// TwinCAT 3 PLC project PRG_B_IO
// Title: B_IO
// Company: RafalOS
// Author: Rafał Osajda
// ProjectVersion: 0.0.0.7
// ProgramVersion: 3.1.4024.0
// libraries:
//   B_Base, * (RafalOS)
//   Tc2_Standard, * (Beckhoff Automation GmbH)
//   Tc2_System, * (Beckhoff Automation GmbH)
//   Tc3_Module, * (Beckhoff Automation GmbH)
// project tree:
//   / PlcTask.TcTTO (not stored)
//   POUs Compilation/ PRG_Compilation.TcPOU (not stored)
//   POUs/Electrovalve/ E_IOElectrovalveAction.TcDUT (not stored), E_IOElectrovalveType.TcDUT (not stored), FB_IOElectrovalve.TcPOU, FB_IOElectrovalve_3on2_NC.TcPOU (not stored), FB_IOElectrovalve_3on2_NO.TcPOU (not stored), FB_IOElectrovalve_5on2_1Coil.TcPOU, FB_IOElectrovalve_5on2_2Coil.TcPOU (not stored), FB_IOElectrovalve_5on3_2Coil_Vented.TcPOU (not stored), FB_IOElectrovalve_5on3_2Coil_Infected.TcPOU (not stored), ITF_IOElectrovalve.TcIO, ITF_IOElectrovalve_HMI_Init.TcIO (not stored), ITF_IOElectrovalve_HMI_Connector.TcIO
//   POUs/Sensor/ E_IOSensorType.TcDUT, FB_IOSensor.TcPOU (not stored), FB_IOSensor_NC.TcPOU, FB_IOSensor_NO.TcPOU, FB_IOSensor_NO_2InRow.TcPOU, ITF_IOSensor.TcIO (not stored), ITF_IOSensor_HMI_Init.TcIO (not stored), ITF_IOSensor_HMI_Connector.TcIO (not stored)
//   POUs/LampkaRozszerzona/ FB_IOLampBlinking.TcPOU, ITF_IOLampBlinking.TcIO
//   POUs/Lampka/ FB_IOLamp.TcPOU (not stored), ITF_IOLamp.TcIO
//   POUs/Przyciski/ FB_IOButton.TcPOU (not stored), FB_IOButton_NC.TcPOU (not stored), FB_IOButton_NO.TcPOU (not stored), ITF_IOButton.TcIO

// ---- POUs/Sensor/E_IOSensorType.TcDUT
{attribute 'qualified_only'}
{attribute 'strict'}
TYPE E_IOSensorType :
(
	NO 		:= 0,
	NC		:= 1,
	NOx2	:= 2
);
END_TYPE

// ---- POUs/Electrovalve/ITF_IOElectrovalve.TcIO
(*
	RJM Maszyny sp. z o.o.
	autor 	: Rafał Osajda
	data	: 21.02.2024
	TC		: 3.1 4024.54
	wersja	: 0.0.1.0	: pełna obsługa

	Obsługa elektrozaworu do sterowania siłownikiem pneumatycznym
*)
INTERFACE ITF_IOElectrovalve EXTENDS ITF_BaseComponent

(*
	RJM Maszyny sp. z o.o.
	autor 	: Rafał Osajda
	data	: 21.02.2024
	TC		: 3.1 4024.54
	wersja	: 0.0.1.0	: pełna obsługa

	Ustawienie odpowiednich wyjść
*)
METHOD Contol : BOOL
VAR_INPUT
	eAction									: E_IOElectrovalveAction;
END_VAR
END_METHOD

END_INTERFACE

// ---- POUs/Electrovalve/ITF_IOElectrovalve_HMI_Connector.TcIO
INTERFACE ITF_IOElectrovalve_HMI_Connector EXTENDS ITF_BaseComponent_HMI_Connector

METHOD PUBLIC GetElectrovalveType : E_IOElectrovalveType
VAR_INPUT
END_VAR
END_METHOD

METHOD PUBLIC GetElectrovalveTypeToString : STRING
END_METHOD

METHOD IsActiveCoilA : BOOL
VAR_INPUT
END_VAR
END_METHOD

METHOD IsActiveCoilB : BOOL
VAR_INPUT
END_VAR
END_METHOD

END_INTERFACE

// ---- POUs/LampkaRozszerzona/ITF_IOLampBlinking.TcIO
INTERFACE ITF_IOLampBlinking EXTENDS ITF_IOLamp

(*			
	EVERDE sp. z o.o.
	Rafał Osajda		31.01.2025		TC 4026.13		wer. 0.0.0.1
	Sterowanie działem ipulsatora 
*)
METHOD PUBLIC SetBlink
VAR_INPUT
	bIN				: bool;
END_VAR
END_METHOD

(*			
	EVERDE sp. z o.o.
	Rafał Osajda		31.01.2025		TC 4026.13		wer. 0.0.0.1
	Ustawia czas zgaszonej lampki
*)
METHOD PUBLIC SetTimeOff
VAR_INPUT
	rIN					: REAL;
END_VAR
END_METHOD

(*			
	EVERDE sp. z o.o.
	Rafał Osajda		31.01.2025		TC 4026.13		wer. 0.0.0.1
	
*)
METHOD PUBLIC SetTimeOn
VAR_INPUT
	rIN						: REAL;
END_VAR
END_METHOD

METHOD PUBLIC SetWork
VAR_INPUT
	bShine		: BOOL;
	bBlink		: BOOL;
	rTimeOn		: REAL;
	rTimeOff	: REAL;
END_VAR
END_METHOD

END_INTERFACE

// ---- POUs/Lampka/ITF_IOLamp.TcIO
INTERFACE ITF_IOLamp EXTENDS ITF_BaseComponent

(*			
	EVERDE sp. z o.o.
	Rafał Osajda		05.02.2025		TC 4026.13		wer. 0.0.0.1
	Sterowanie swieceniem lampki - włącz/wyłącz
*)
METHOD Control
VAR_INPUT
	bIN						: BOOL;
END_VAR
END_METHOD

(*			
	EVERDE sp. z o.o.
	Rafał Osajda		05.02.2025		TC 4026.13		wer. 0.0.0.1
	Zwraca czy lampka wlaczona
*)
METHOD IsActive : BOOL
END_METHOD

(*			
	EVERDE sp. z o.o.
	Rafał Osajda		05.02.2025		TC 4026.13		wer. 0.0.0.1
	Wylacza lampke
*)
METHOD SetOff
END_METHOD

(*			
	EVERDE sp. z o.o.
	Rafał Osajda		05.02.2025		TC 4026.13		wer. 0.0.0.1
	Wlacza lampke
*)
METHOD SetOn
END_METHOD

END_INTERFACE

// ---- POUs/Przyciski/ITF_IOButton.TcIO
INTERFACE ITF_IOButton EXTENDS ITF_BaseComponent

METHOD PUBLIC GetRisingEdgePressed : BOOL
VAR_INPUT
END_VAR
END_METHOD

(*			
	EVERDE sp. z o.o.
	Rafał Osajda		31.01.2025		TC 4026.13		wer. 0.0.0.1
	Zwraca stan przycisku
*)
METHOD IsPressed : BOOL
END_METHOD

END_INTERFACE

// ---- POUs/Sensor/FB_IOSensor_NC.TcPOU
(*			
	EVERDE sp. z o.o.
	Rafał Osajda		22.01.2025		TC 4026.13		wer. 0.0.0.1
	B_Baza dla czujników binarnych styk normalnie zamkniety 	
*)
FUNCTION_BLOCK FB_IOSensor_NC EXTENDS FB_IOSensor
VAR
END_VAR

METHOD FB_init : BOOL
VAR_INPUT
	bInitRetains : BOOL; // if TRUE, the retain variables are initialized (warm start / cold start)
	bInCopyCode : BOOL;  // if TRUE, the instance afterwards gets moved into the copy code (online change)
END_VAR
THIS^.eType		:= E_IOSensorType.NC;
END_METHOD

(*			
	EVERDE sp. z o.o.
	Rafał Osajda		05.02.2025		TC 4026.13		wer. 0.0.0.1
	Zwraca aktualny stan czujnika
*)
METHOD IsActive : BOOL
IsActive				:= NOT THIS^.bContact;
END_METHOD

END_FUNCTION_BLOCK

// ---- POUs/Sensor/FB_IOSensor_NO.TcPOU
(*			
	EVERDE sp. z o.o.
	Rafał Osajda		22.01.2025		TC 4026.13		wer. 0.0.0.1
	B_Baza dla czujników binarnych styk normalnie otwarty 	
*)
FUNCTION_BLOCK FB_IOSensor_NO EXTENDS FB_IOSensor
VAR
END_VAR

METHOD FB_init : BOOL
VAR_INPUT
	bInitRetains : BOOL; // if TRUE, the retain variables are initialized (warm start / cold start)
	bInCopyCode : BOOL;  // if TRUE, the instance afterwards gets moved into the copy code (online change)
END_VAR
THIS^.eType		:= E_IOSensorType.NO;
END_METHOD

(*			
	EVERDE sp. z o.o.
	Rafał Osajda		05.02.2025		TC 4026.13		wer. 0.0.0.1
	Zwraca aktualny stan czujnika
*)
METHOD IsActive : BOOL
IsActive			:= THIS^.bContact;
END_METHOD

END_FUNCTION_BLOCK

// ---- POUs/Sensor/FB_IOSensor_NO_2InRow.TcPOU
(*
	EVERDE sp. z o.o.
	Rafał Osajda
	18.09.2024
	TC3 4026.10
	Obsługa czujników cyforwych NO połączonych szerogowo
*)
FUNCTION_BLOCK FB_IOSensor_NO_2InRow EXTENDS FB_IOSensor_NO
VAR
	bContact2							AT %I*	: BOOL;		//fizyczne wejście z czujnika
END_VAR

METHOD FB_init : BOOL
VAR_INPUT
	bInitRetains : BOOL; // if TRUE, the retain variables are initialized (warm start / cold start)
	bInCopyCode : BOOL;  // if TRUE, the instance afterwards gets moved into the copy code (online change)
END_VAR
THIS^.eType		:= E_IOSensorType.NOx2;
END_METHOD

(*			
	EVERDE sp. z o.o.
	Rafał Osajda		05.02.2025		TC 4026.13		wer. 0.0.0.1
	Zwraca aktualny stan czujnika
*)
METHOD IsActive : BOOL
IsActive				:=  THIS^.bContact AND THIS^.bContact2;
END_METHOD

END_FUNCTION_BLOCK

// ---- POUs/Electrovalve/FB_IOElectrovalve.TcPOU
(*
	RJM Maszyny sp. z o.o.
	autor 	: Rafał Osajda
	data	: 02.02.2024
	TC		: 3.1 4024.54
	wersja	: 0.0.1.0	: pełna obsługa

	Obsługa elektrozaworu do sterowania siłownikiem pneumatycznym. FB bazowy dla pozostałych rodzajów elektrozaworów
*)
FUNCTION_BLOCK ABSTRACT FB_IOElectrovalve EXTENDS FB_BaseComponent IMPLEMENTS  ITF_IOElectrovalve, ITF_IOElectrovalve_HMI_Init
VAR
	bCoilA							AT %Q*	: BOOL;
	bCoilB							AT %Q*	: BOOL;
	eType									: E_IOElectrovalveType;
END_VAR

(*
	RJM Maszyny sp. z o.o.
	autor 	: Rafał Osajda
	data	: 21.02.2024
	TC		: 3.1 4024.54
	wersja	: 0.0.1.0	: pełna obsługa

	Ustawienie odpowiednich wyjść
*)
METHOD Contol : BOOL
VAR_INPUT
	eAction	: E_IOElectrovalveAction;
END_VAR
END_METHOD

METHOD PUBLIC GetElectrovalveType : E_IOElectrovalveType
VAR_INPUT
END_VAR
GetElectrovalveType			:= THIS^.eType;
END_METHOD

METHOD PUBLIC GetElectrovalveTypeToString : STRING
VAR CONSTANT
	arrType		: ARRAY [0..5] OF STRING := ['NC_3na2', 'NO_3na2', 'C1_5na2', 'C2_5na2', 'C2_5na3O', 'C2_5na3Z'];
END_VAR
GetElectrovalveTypeToString			:= arrType [TO_INT (THIS^.eType)];
END_METHOD

METHOD IsActiveCoilA : BOOL
VAR_INPUT
END_VAR
IsActiveCoilA			:= THIS^.bCoilA;
END_METHOD

METHOD IsActiveCoilB : BOOL
VAR_INPUT
END_VAR
IsActiveCoilB			:= THIS^.bCoilB;
END_METHOD

END_FUNCTION_BLOCK

// ---- POUs/Electrovalve/FB_IOElectrovalve_5on2_1Coil.TcPOU
(*
	RJM Maszyny sp. z o.o.
	autor 	: Rafał Osajda
	data	: 02.02.2024
	TC		: 3.1 4024.54
	wersja	: 0.0.1.0	: pełna obsługa

	Obsługa elektrozaworu do sterowania siłownikiem pneumatycznym.sterowanie 5 na 2 1 cewka
*)
FUNCTION_BLOCK FB_IOElectrovalve_5on2_1Coil EXTENDS FB_IOElectrovalve

(*
	RJM Maszyny sp. z o.o.
	autor 	: Rafał Osajda
	data	: 21.02.2024
	TC		: 3.1 4024.54
	wersja	: 0.0.1.0	: pełna obsługa

	Ustawienie odpowiednich wyjść
*)
METHOD Contol : BOOL
VAR_INPUT
	eAction	: E_IOElectrovalveAction;
END_VAR
CASE eAction OF
	E_IOElectrovalveAction.e_EV_Out4_Deactive	:
		bCoilA								:= FALSE;
	E_IOElectrovalveAction.e_EV_OUT4_Active	:
		bCoilA								:= TRUE;
	E_IOElectrovalveAction.e_EV_ToStart	:
		bCoilA								:= FALSE;
	E_IOElectrovalveAction.e_EV_ToEnd		:
		bCoilA								:= TRUE;
	E_IOElectrovalveAction.e_EV_Reset			:
		bCoilA								:= FALSE;
END_CASE
THIS^.bCoilB								:= FALSE;
END_METHOD

METHOD FB_init : BOOL
VAR_INPUT
	bInitRetains : BOOL; // if TRUE, the retain variables are initialized (warm start / cold start)
	bInCopyCode : BOOL;  // if TRUE, the instance afterwards gets moved into the copy code (online change)
END_VAR
THIS^.eType			:= E_IOElectrovalveType.C1_5na2;
END_METHOD

END_FUNCTION_BLOCK

// ---- POUs/LampkaRozszerzona/FB_IOLampBlinking.TcPOU
(*			
	EVERDE sp. z o.o.
	Rafał Osajda		16.07.2025		TC 4024.66
	Lampka rozszerzona o moduł FB_Impuls co integruje w niej możlwiość mgania lub świecenie ciągłego
*)
FUNCTION_BLOCK FB_IOLampBlinking EXTENDS FB_IOLamp IMPLEMENTS ITF_IOLampBlinking
VAR
	fbImpulse				: FB_BaseImpulse;
END_VAR

(*			
	EVERDE sp. z o.o.
	Rafał Osajda		05.02.2025		TC 4026.13		wer. 0.0.0.1
	Sterowanie swieceniem lampki - włącz/wyłącz
*)
METHOD Control
VAR_INPUT
	bIN	: BOOL;
END_VAR
IF (bIN) THEN
	THIS^.fbImpulse.SetExecuteOn ();
ELSE
	THIS^.fbImpulse.SetExecuteOff ();
END_IF
END_METHOD

(*			
	EVERDE sp. z o.o.
	Rafał Osajda		27.03.2025		TC 4024.66
	Wywolanie co cykl operacji 
*)
METHOD PUBLIC ExecuteEveryCycle_Operation
VAR_INPUT
END_VAR
SUPER^.ExecuteEveryCycle_Operation ();

THIS^.fbImpulse ();
END_METHOD

(*			
	EVERDE sp. z o.o.
	Rafał Osajda		27.03.2025		TC 4024.66
	Aktualizacja flag 
*)
METHOD PUBLIC ExecuteEveryCycle_Status
VAR_INST
END_VAR
SUPER^.ExecuteEveryCycle_Status ();

THIS^.bOut		:= THIS^.fbImpulse.GetExit ();
END_METHOD

(*			
	EVERDE sp. z o.o.
	Rafał Osajda		31.01.2025		TC 4026.13		wer. 0.0.0.1
	Sterowanie działem ipulsatora 
*)
METHOD PUBLIC SetBlink
VAR_INPUT
	bIN				: bool;
END_VAR
THIS^.fbImpulse.SetFlashing (bIN	:= bIN);
END_METHOD

(*			
	EVERDE sp. z o.o.
	Rafał Osajda		05.02.2025		TC 4026.13		wer. 0.0.0.1
	Wylacza lampke
*)
METHOD SetOff
THIS^.fbImpulse.SetExecuteOff ();
END_METHOD

(*			
	EVERDE sp. z o.o.
	Rafał Osajda		05.02.2025		TC 4026.13		wer. 0.0.0.1
	Wlacza lampke - praca ciągła
*)
METHOD SetOn
THIS^.fbImpulse.SetExecuteOn ();
END_METHOD

METHOD PUBLIC SetShine
VAR_INPUT
	bIN				: BOOL;
END_VAR
IF (bIN) THEN
	THIS^.fbImpulse.SetExecuteOn ();
ELSE
	THIS^.fbImpulse.SetExecuteOff ();
END_IF
END_METHOD

(*			
	EVERDE sp. z o.o.
	Rafał Osajda		31.01.2025		TC 4026.13		wer. 0.0.0.1
	Ustawia czas zgaszonej lampki
*)
METHOD PUBLIC SetTimeOff
VAR_INPUT
	rIN					: REAL;
END_VAR
THIS^.fbImpulse.SetTimeOff (rIN	:= rIN);
END_METHOD

(*			
	EVERDE sp. z o.o.
	Rafał Osajda		31.01.2025		TC 4026.13		wer. 0.0.0.1
	
*)
METHOD PUBLIC SetTimeOn
VAR_INPUT
	rIN						: REAL;
END_VAR
THIS^.fbImpulse.SetTimeOn (rIN	:= rIN);
END_METHOD

METHOD PUBLIC SetWork
VAR_INPUT
	bShine		: BOOL;
	bBlink		: BOOL;
	rTimeOn		: REAL;
	rTimeOff	: REAL;
END_VAR
THIS^.fbImpulse.SetTimeOn (rIN := rTimeOn);
THIS^.fbImpulse.SetTimeOff (rIN := rTimeOff);
THIS^.SetShine (bIN	:= bShine);
THIS^.SetBlink (bIN := bBlink);
END_METHOD

END_FUNCTION_BLOCK
